FUNCTION adc_to_float_pv : LREAL
VAR_INPUT
	i			: LREAL;
	pv_max		: LREAL;
	pv_min		: LREAL;
	i_max		: LREAL;
	i_min		: LREAL;
END_VAR
VAR
	m			: LREAL;
END_VAR


m := (pv_max-pv_min)/(i_max-i_min);

adc_to_float_pv	:=	m*(i-i_min) + pv_min;

END_FUNCTION

(* stored: Version 1.1.0.1, ProductVersion 3.1.0.36
   POU adc_to_float_pv: Id {d8bea1e0-e369-4414-bffa-3400a28a10d5}, SpecialFunc None *)
